FUNCTION_BLOCK RF_TRIG (* Basic Function Block Type *)
  (* Standard: 61499-2 *)
  (* Version 0.0, 08.09.2011, herrric, nxtControl GmbH, Template *)
  PACKAGE Loytec.Automation;
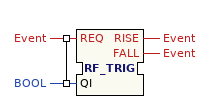
  EVENT_INPUT
    REQ WITH QI; (* Normal Execution Request *)
  END_EVENT
  EVENT_OUTPUT
    RISE;
    FALL;
  END_EVENT
  VAR_INPUT
    QI : BOOL; (* Input event qualifier *)
  END_VAR
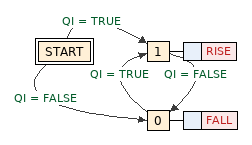
  EC_STATES
    START; (* Initial State *)
    1 : -> RISE; (* Initialization *)
    0 : -> FALL; (* Normal execution *)
  END_STATES
  EC_TRANSITIONS
    0 TO 1 := QI = TRUE;
    1 TO 0 := QI = FALSE;
    START TO 1 := QI = TRUE;
    START TO 0 := QI = FALSE;
  END_TRANSITIONS
  ALGORITHM INIT IN ST: (* Initialization algorithm *)
;
  END_ALGORITHM
  ALGORITHM REQ IN ST: (* Normally executed algorithm *)
;
  END_ALGORITHM
END_FUNCTION_BLOCK
